// TIA Portal project "Project_asynchronousmotor_stardeltastarting_sim" (V16)

(* hardware
DEVICE "S7-1200 station_1"  S7-1200 Station
   slot 0: "Rack_0"  S7-1200 Rack  Rack  V1.0
   slot 1: "PLC_1"  CPU 1212C DC/DC/Rly  6ES7 212-1HE40-0XB0  V4.4
   slot 2: "DQ 8x24VDC _1"  SM 1222 DQ8 x 24VDC  6ES7 222-1BF32-0XB0  V2.0
   slot 3: "DI 4x24VDC_1"  DI4 signal board (200 kHz)  6ES7 221-3BD30-0XB0  V1.0
*)

// ===== PLC "PLC_1"  CPU 1212C DC/DC/Rly =====

VAR_GLOBAL   // PLC tag table "Default tag table"
   ""START BUT"" AT %I4.0 : Bool;
   ""STOP BUT"" AT %I4.1 : Bool;
   ""ANA KONT"" AT %Q8.0 : Bool;
   ""YILDIZ KONT"" AT %Q8.1 : Bool;
   ""UCGEN KONT"" AT %Q8.2 : Bool;
END_VAR